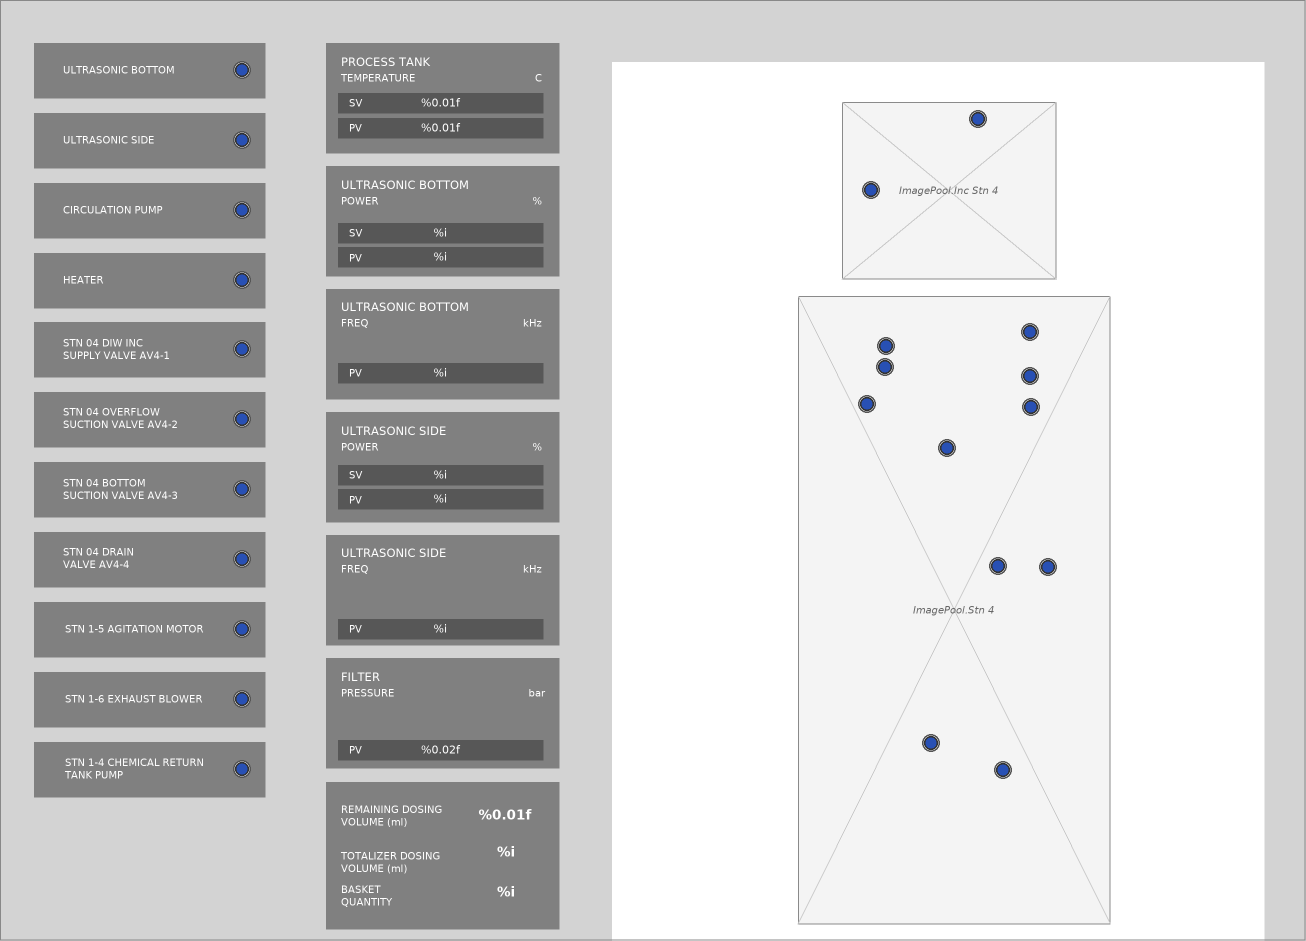
VISUALIZATION Auto_Station04  // 1306x941
    Rectangle (0,0 1306x875)
    RoundedRectangle (34,43 231x55)
    Label (60,62 163x16), "ULTRASONIC BOTTOM"
    Lamp1 (232,60 20x20), variable: ARdsMAP_HmiVariableStn[4].bProTankUsBtm_IND, style: Lamp-Lamp1-Blue
    RoundedRectangle (34,183 231x55)
    Label (60,202 151x16), "CIRCULATION PUMP"
    Lamp1 (232,200 20x20), variable: ARdsMAP_HmiVariableStn[4].bProTankPump_IND, style: Lamp-Lamp1-Blue
    RoundedRectangle (34,253 231x55)
    Label (60,272 151x16), "HEATER"
    Lamp1 (232,270 20x20), variable: ARdsMAP_HmiVariableStn[4].bProTankHeater_IND, style: Lamp-Lamp1-Blue
    RoundedRectangle (34,113 231x55)
    Label (60,132 163x16), "ULTRASONIC SIDE"
    Lamp1 (232,130 20x20), variable: ARdsMAP_HmiVariableStn[4].bProTankUsSide_IND, style: Lamp-Lamp1-Blue
    RoundedRectangle (34,322 231x55)
    Label (60,336 151x27), "STN 04 DIW INC SUPPLY VALVE AV4-1"
    Lamp1 (232,339 20x20), variable: ARdsMAP_HmiVariableStn[4].bValve01_IND, style: Lamp-Lamp1-Blue
    RoundedRectangle (34,392 231x55)
    Lamp1 (232,409 20x20), variable: ARdsMAP_HmiVariableStn[4].bValve02_IND, style: Lamp-Lamp1-Blue
    Label (60,405 168x27), "STN 04 OVERFLOW SUCTION VALVE AV4-2"
    RoundedRectangle (34,462 231x55)
    Label (60,476 151x27), "STN 04 BOTTOM SUCTION VALVE AV4-3"
    Lamp1 (232,479 20x20), variable: ARdsMAP_HmiVariableStn[4].bValve03_IND, style: Lamp-Lamp1-Blue
    RoundedRectangle (34,532 231x55)
    Lamp1 (232,549 20x20), variable: ARdsMAP_HmiVariableStn[4].bValve04_IND, style: Lamp-Lamp1-Blue
    Label (60,545 168x27), "STN 04 DRAIN VALVE AV4-4"
    RoundedRectangle (34,602 231x55)
    Label (62,611 160x36), "STN 1-5 AGITATION MOTOR"
    Lamp1 (232,619 20x20), variable: ARdsMAP_HmiVariableGeneral.bProTankAgitationMotor_IND, style: Lamp-Lamp1-Blue
    RoundedRectangle (34,672 231x55)
    Label (62,681 160x36), "STN 1-6 EXHAUST BLOWER"
    Lamp1 (232,689 20x20), variable: ARdsMAP_HmiVariableGeneral.bExhaustBlower_IND, style: Lamp-Lamp1-Blue
    RoundedRectangle (34,742 231x55)
    Label (62,751 160x36), "STN 1-4 CHEMICAL RETURN TANK PUMP"
    Lamp1 (232,759 20x20), variable: ARdsMAP_HmiVariableGeneral.bProTankPump_IND, style: Lamp-Lamp1-Blue
    Rectangle (612,62 652x879)
    Image (798,296 312x628), image: ImagePool.Stn 4
    Lamp1 (937,438 20x20), variable: ARdsMAP_HmiVariableStn[4].bProTankUsBtm_IND, style: Lamp-Lamp1-Blue
    Lamp1 (921,733 20x20), variable: ARdsMAP_HmiVariableStn[4].bProTankPump_IND, style: Lamp-Lamp1-Blue
    Lamp1 (875,357 20x20), variable: ARdsMAP_HmiVariableStn[4].bProTankHeater_IND, style: Lamp-Lamp1-Blue
    Lamp1 (857,394 20x20), variable: ARdsMAP_HmiVariableStn[4].bProTankUsSide_IND, style: Lamp-Lamp1-Blue
    Lamp1 (1038,557 20x20), variable: ARdsMAP_HmiVariableStn[4].bValve02_IND, style: Lamp-Lamp1-Blue
    Lamp1 (993,760 20x20), variable: ARdsMAP_HmiVariableStn[4].bValve04_IND, style: Lamp-Lamp1-Blue
    Lamp1 (988,556 20x20), variable: ARdsMAP_HmiVariableStn[4].bValve03_IND, style: Lamp-Lamp1-Blue
    Lamp1 (1020,322 20x20), variable: ARdsMAP_HmiVariableStn[4].bOverflowMaxLevel_IND, style: Lamp-Lamp1-Blue
    Lamp1 (876,336 20x20), variable: ARdsMAP_HmiVariableStn[4].bProcessTankMinLevel_IND, style: Lamp-Lamp1-Blue
    Lamp1 (1020,366 20x20), variable: ARdsMAP_HmiVariableStn[4].bOverflowMinLevel_IND, style: Lamp-Lamp1-Blue
    Lamp1 (1021,397 20x20), variable: ARdsMAP_HmiVariableStn[4].bProTankUsSide_IND, style: Lamp-Lamp1-Blue
    Image (842,102 214x177), image: ImagePool.Inc Stn 4
    Lamp1 (968,109 20x20), variable: ARdsMAP_HmiVariableStn[4].bValve01_IND, style: Lamp-Lamp1-Blue
    Lamp1 (861,180 20x20), variable: ARdsMAP_HmiVariableStn[4].bDosingPump_IND, style: Lamp-Lamp1-Blue
    RoundedRectangle (326,43 233x110)
    Label (338,54 150x16), "PROCESS TANK"
    Label (338,67 99x22), "TEMPERATURE"
    Label (516,67 29x22), "C"
    Rectangle (338,93 205x20), "%0.01f", text variable: ARrStnTempSV[4]
    Label (346,92 22x22), "SV"
    Rectangle (338,118 205x20), "%0.01f", text variable: ARrStnTempPV[4]
    Label (346,117 22x22), "PV"
    RoundedRectangle (326,166 233x110)
    Label (338,177 150x16), "ULTRASONIC BOTTOM"
    Label (338,190 99x22), "POWER"
    Label (516,190 29x22), "%"
    Rectangle (338,223 205x20), "%i", text variable: DSWeberEnclosure[2].DSWeberGenerator[2].IN_iTargetPowerPercentSetPoint
    Label (346,222 22x22), "SV"
    Rectangle (338,247 205x20), "%i", text variable: ARiStnUSBtmAPv[4]
    Label (346,247 22x22), "PV"
    RoundedRectangle (326,658 233x110)
    Label (338,669 150x16), "FILTER"
    Label (338,682 99x22), "PRESSURE"
    Label (516,682 32x22), "bar"
    Rectangle (338,740 205x20), "%0.02f", text variable: ARrStnFilterPressurePV[4]
    Label (346,739 22x22), "PV"
    RoundedRectangle (326,289 233x110)
    Label (338,312 99x22), "FREQ"
    Label (338,299 150x16), "ULTRASONIC BOTTOM"
    Label (516,312 29x22), "kHz"
    Rectangle (338,363 205x20), "%i", text variable: ARiStnUSBtmAFreqPv[4]
    Label (346,362 22x22), "PV"
    RoundedRectangle (326,782 233x147)
    Label (338,845 118x35), "TOTALIZER DOSING VOLUME (ml)"
    Label (338,802 118x28), "REMAINING DOSING VOLUME (ml)"
    Rectangle (464,801 82x28), "%0.01f", text variable: ARDSProminentDosingHMI[4].Out_rRemainedDosingVolume_ml
    Rectangle (465,838 82x28), "%i", text variable: ARDSProminentDosingHMI[4].Out_iDosingTotalizer_ml
    Label (338,882 118x28), "BASKET QUANTITY"
    Rectangle (465,878 82x28), "%i", text variable: ARDSProminentDosingHMI[4].Out_iBasketQtyBeforeAutoDosingPV
    RoundedRectangle (326,412 233x110)
    Label (338,423 150x16), "ULTRASONIC SIDE"
    Label (338,436 99x22), "POWER"
    Label (516,436 29x22), "%"
    Rectangle (338,465 205x20), "%i", text variable: DSWeberEnclosure[2].DSWeberGenerator[1].IN_iTargetPowerPercentSetPoint
    Label (346,464 22x22), "SV"
    Rectangle (338,489 205x20), "%i", text variable: ARiStnUSSideAPv[4]
    Label (346,489 22x22), "PV"
    RoundedRectangle (326,535 233x110)
    Label (338,558 99x22), "FREQ"
    Label (338,545 150x16), "ULTRASONIC SIDE"
    Label (516,558 29x22), "kHz"
    Rectangle (338,619 205x20), "%i", text variable: ARiStnUSSideAFreqPv[4]
    Label (346,618 22x22), "PV"
END_VISUALIZATION

(* stored: Version 1.1.0.1, ProductVersion 3.1.4024.12
   Visu Auto_Station04: Id {d52b36e3-768f-4f57-9eaa-1a5f863bd053} *)
